// Mitsubishi GX Works2 project: memoryIO   PLC: Q02/Q02H

PROGRAM wordCTRL
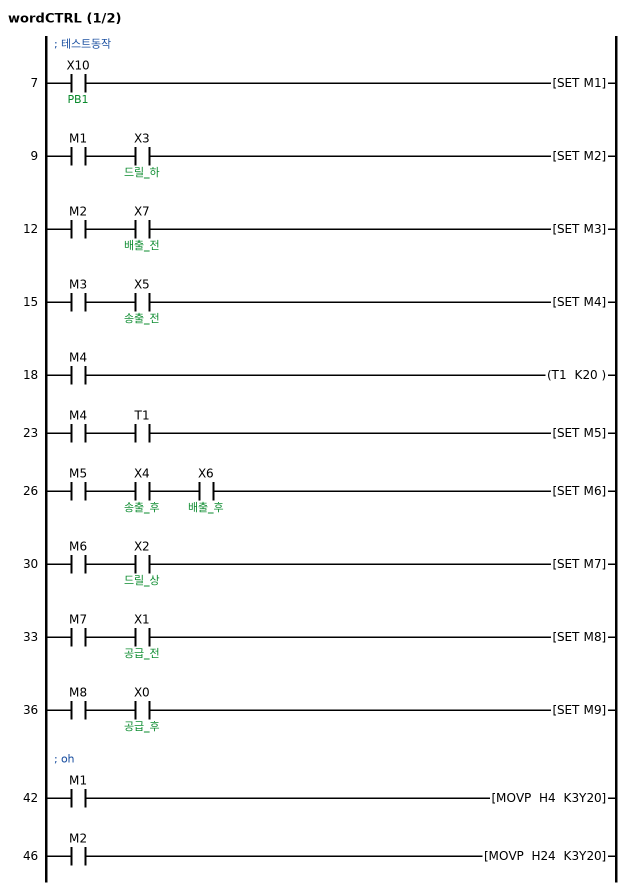
; 테스트동작
7     LD      X10  ; PB1
      SET     M1
9     LD      M1
      AND     X3  ; 드릴_하
      SET     M2
12    LD      M2
      AND     X7  ; 배출_전
      SET     M3
15    LD      M3
      AND     X5  ; 송출_전
      SET     M4
18    LD      M4
      OUT     T1 K20
23    LD      M4
      AND     T1
      SET     M5
26    LD      M5
      AND     X4  ; 송출_후
      AND     X6  ; 배출_후
      SET     M6
30    LD      M6
      AND     X2  ; 드릴_상
      SET     M7
33    LD      M7
      AND     X1  ; 공급_전
      SET     M8
36    LD      M8
      AND     X0  ; 공급_후
      SET     M9
; oh
42    LD      M1
      MOVP    H4 K3Y20  ; 공급_전
46    LD      M2
      MOVP    H24 K3Y20
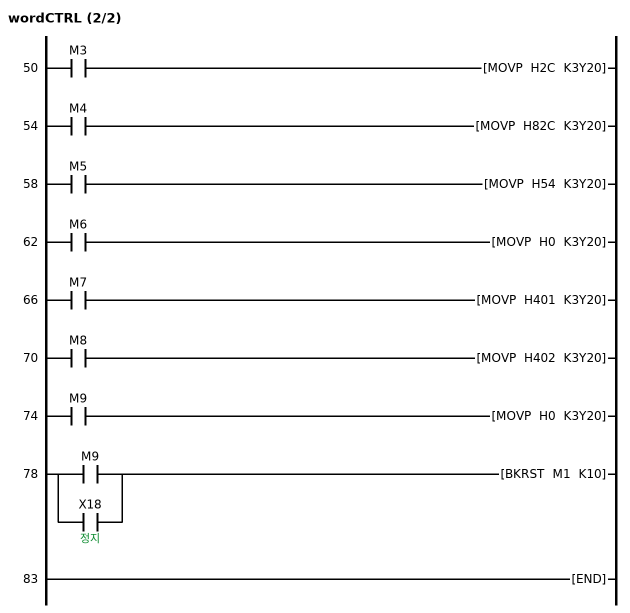
50    LD      M3
      MOVP    H2C K3Y20
54    LD      M4
      MOVP    H82C K3Y20
58    LD      M5
      MOVP    H54 K3Y20
62    LD      M6
      MOVP    H0 K3Y20
66    LD      M7
      MOVP    H401 K3Y20
70    LD      M8
      MOVP    H402 K3Y20
74    LD      M9
      MOVP    H0 K3Y20
78    LD      M9
      OR      X18  ; 정지
      BKRST   M1 K10
83    END
END_PROGRAM

PROGRAM batchIO
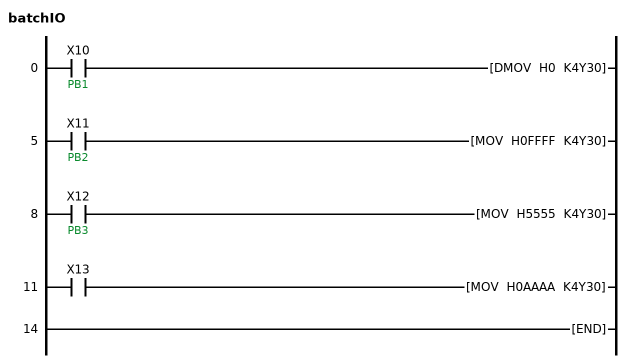
0     LD      X10  ; PB1
      DMOV    H0 K4Y30
5     LD      X11  ; PB2
      MOV     H0FFFF K4Y30
8     LD      X12  ; PB3
      MOV     H5555 K4Y30
11    LD      X13
      MOV     H0AAAA K4Y30
14    END
END_PROGRAM

// device comments not shown above
X8  ; 매거진
X9  ; 비금속
X0A  ; 금속
Y21  ; 공급_후
Y22  ; 드릴_전
Y23  ; 송출_전
Y24  ; 송출_후
Y25  ; 배출_전
Y26  ; 배출_후
Y27  ; 컨베이어
Y28  ; 가공도
Y29  ; 적색
Y2A  ; 황색
Y2B  ; 녹색
